{attribute 'qualified_only'}
{attribute 'strict'}
TYPE E_ReadWriteStep :
(
	SEND,
	AWAIT_RESPONSE
);
END_TYPE

(* stored: Version 1.1.0.1, ProductVersion 3.1.4024.13
   DUT E_ReadWriteStep: Id {1eed6091-67d3-0520-37f3-26158e8fc93d} *)
